# EPICS substitutions: iocBoot/obsolete/ioc13sdd1/4element.substitutions
file "$(DXP)/db/dxpSystem.template" {
{P=13SDD1:, IO="@asyn(DXP1,0)"}
}

file "$(DXP)/db/dxpMED.template" {
{P=13SDD1:, DETALL="@asyn(DXP1,4,1)"}
}

file "$(DXP)/db/dxpMapping.template" {
{P=13SDD1:, IO="@asyn(DXP1,0)"}
}

# DXP parameters
file "$(DXP)/db/dxpHighLevel.template"
{
pattern
{       P,       R,           IO}
{13SDD1:,    dxp1:,  "@asyn(DXP1,0,1)"}
{13SDD1:,    dxp2:,  "@asyn(DXP1,1,1)"}
{13SDD1:,    dxp3:,  "@asyn(DXP1,2,1)"}
{13SDD1:,    dxp4:,  "@asyn(DXP1,3,1)"}
}

# Low-level parameters
file "$(DXP)/db/dxpLowLevel.template"
{
pattern
{       P,       R,        IO}
{13SDD1:,    dxp1:,  "@asyn(DXP1,0,1)"}
{13SDD1:,    dxp2:,  "@asyn(DXP1,1,1)"}
{13SDD1:,    dxp3:,  "@asyn(DXP1,2,1)"}
{13SDD1:,    dxp4:,  "@asyn(DXP1,3,1)"}
}

# SCA parameters
file "$(DXP)/db/dxpSCA_16.template"
{
pattern
{       P,       R,          IO}
{13SDD1:,    dxp1:,  "@asyn(DXP1,0,1)"}
{13SDD1:,    dxp2:,  "@asyn(DXP1,1,1)"}
{13SDD1:,    dxp3:,  "@asyn(DXP1,2,1)"}
{13SDD1:,    dxp4:,  "@asyn(DXP1,3,1)"}
}

file "$(MCA)/db/simple_mca.db"
{
pattern
{       P,      M,       DTYP,               INP,  PREC,    CHANS}
{13SDD1:,   mca1,  "asynMCA",   "@asyn(DXP1,0)",     2,     2048}
{13SDD1:,   mca2,  "asynMCA",   "@asyn(DXP1,1)",     2,     2048}
{13SDD1:,   mca3,  "asynMCA",   "@asyn(DXP1,2)",     2,     2048}
{13SDD1:,   mca4,  "asynMCA",   "@asyn(DXP1,3)",     2,     2048}
}

file "$(ASYN)/db/asynRecord.db"
{
pattern
{       P,    R,  PORT,   ADDR,  IMAX,  OMAX}
{13SDD1:, Asyn,  DXP1,      0,    80,    80}
}
